PROGRAM P_Simulator
VAR
	fbCraneSimulator : FB_CraneSimulator;
END_VAR

fbCraneSimulator(
	ssMethodType := BOOL_TO_SINT(G_Simulator.bSimulatorOn),
	uDCV := G_Work.fControlOutputNormalized,
	ppbar => G_Simulator.fPistonSidePressure,
	prbar => G_Simulator.fRodSidePressure,
	xm => G_Simulator.fPistonPosition
);

END_PROGRAM

(* stored: Version 1.1.0.1, ProductVersion 3.1.4024.10
   POU P_Simulator: Id {536492b7-da96-4ec3-8126-8b196493af0f}, SpecialFunc None *)
